           #Q_L2_max := #ZQ_L2_max / #MILLION / #THOUSAND;
           #Q_L3_max := #ZQ_L3_max / #MILLION / #THOUSAND;
   END_CASE;
   // calculate apparent energy unit     
   CASE #C_E_S_Unit OF
       1:
           IF ((#VEnergy_Meter_Unit[9] = TRUE) OR (#VEnergy_Meter_Unit[10] = TRUE)) THEN
               #S_Energy_Unit := 'kVAh';
               IF (#VEnergy_Meter_Unit[9] = FALSE) THEN
                   #E_Apparent_Rate1_Import := #ZE_Apparent_Rate1_Import / #THOUSAND;
               ELSE
                   #E_Apparent_Rate1_Import := #ZE_Apparent_Rate1_Import;
               END_IF;
               IF (#VEnergy_Meter_Unit[10] = FALSE) THEN
                   #E_Apparent_Rate2_Import := #ZE_Apparent_Rate2_Import / #THOUSAND;
               ELSE
                   #E_Apparent_Rate2_Import := #ZE_Apparent_Rate2_Import;
               END_IF;
           ELSE
               #S_Energy_Unit := 'VAh';
               #E_Apparent_Rate1_Import := #ZE_Apparent_Rate1_Import;
               #E_Apparent_Rate2_Import := #ZE_Apparent_Rate2_Import;
           END_IF;
       2:
           IF ((#VEnergy_Meter_Unit[9] = TRUE) OR (#VEnergy_Meter_Unit[10] = TRUE)) THEN
               #S_Energy_Unit := 'MVAh';
               IF (#VEnergy_Meter_Unit[9] = FALSE) THEN
                   #E_Apparent_Rate1_Import := #ZE_Apparent_Rate1_Import / #MILLION;
               ELSE
                   #E_Apparent_Rate1_Import := #ZE_Apparent_Rate1_Import / #THOUSAND;
               END_IF;
               IF (#VEnergy_Meter_Unit[10] = FALSE) THEN
                   #E_Apparent_Rate2_Import := #ZE_Apparent_Rate2_Import / #MILLION;
               ELSE
                   #E_Apparent_Rate2_Import := #ZE_Apparent_Rate2_Import / #THOUSAND;
               END_IF;
           ELSE
               #S_Energy_Unit := 'kVAh';
               #E_Apparent_Rate1_Import := #ZE_Apparent_Rate1_Import / #THOUSAND;
               #E_Apparent_Rate2_Import := #ZE_Apparent_Rate2_Import / #THOUSAND;
           END_IF;
       3:
           IF ((#VEnergy_Meter_Unit[9] = TRUE) OR (#VEnergy_Meter_Unit[10] = TRUE)) THEN
               #S_Energy_Unit := 'GVAh';
               IF (#VEnergy_Meter_Unit[9] = FALSE) THEN
                   #E_Apparent_Rate1_Import := #ZE_Apparent_Rate1_Import / #MILLION / #THOUSAND;
               ELSE
                   #E_Apparent_Rate1_Import := #ZE_Apparent_Rate1_Import / #MILLION;
               END_IF;
               IF (#VEnergy_Meter_Unit[10] = FALSE) THEN
                   #E_Apparent_Rate2_Import := #ZE_Apparent_Rate2_Import / #MILLION / #THOUSAND;
               ELSE
                   #E_Apparent_Rate2_Import := #ZE_Apparent_Rate2_Import / #MILLION;
               END_IF;
           ELSE
               #S_Energy_Unit := 'MVAh';
               #E_Apparent_Rate1_Import := #ZE_Apparent_Rate1_Import / #MILLION;
               #E_Apparent_Rate2_Import := #ZE_Apparent_Rate2_Import / #MILLION;
           END_IF;
       ELSE:
           IF ((#VEnergy_Meter_Unit[9] = TRUE) OR (#VEnergy_Meter_Unit[10] = TRUE)) THEN
               #S_Energy_Unit := 'TVAh';
               IF (#VEnergy_Meter_Unit[9] = FALSE) THEN
                   #E_Apparent_Rate1_Import := #ZE_Apparent_Rate1_Import / #MILLION / #MILLION;
               ELSE
                   #E_Apparent_Rate1_Import := #ZE_Apparent_Rate1_Import / #MILLION / #THOUSAND;
               END_IF;
               IF (#VEnergy_Meter_Unit[10] = FALSE) THEN
                   #E_Apparent_Rate2_Import := #ZE_Apparent_Rate2_Import / #MILLION / #MILLION;
               ELSE
                   #E_Apparent_Rate2_Import := #ZE_Apparent_Rate2_Import / #MILLION / #THOUSAND;
               END_IF;
           ELSE
               #S_Energy_Unit := 'GVAh';
               #E_Apparent_Rate1_Import := #ZE_Apparent_Rate1_Import / #MILLION / #THOUSAND;
               #E_Apparent_Rate2_Import := #ZE_Apparent_Rate2_Import / #MILLION / #THOUSAND;
           END_IF;
   END_CASE;
   // calculate active energy unit     
   CASE #C_E_P_Unit OF
       1:
           IF ((#VEnergy_Meter_Unit[1] = TRUE) OR (#VEnergy_Meter_Unit[2] = TRUE) OR
               (#VEnergy_Meter_Unit[3] = TRUE) OR (#VEnergy_Meter_Unit[4] = TRUE)) THEN
               #P_Energy_Unit := 'kWh';
               IF (#VEnergy_Meter_Unit[1] = FALSE) THEN
                   #E_Active_Rate1_Import := #ZE_Active_Rate1_Import / #THOUSAND;
               ELSE
                   #E_Active_Rate1_Import := #ZE_Active_Rate1_Import;
               END_IF;
               IF (#VEnergy_Meter_Unit[2] = FALSE) THEN
                   #E_Active_Rate2_Import := #ZE_Active_Rate2_Import / #THOUSAND;
               ELSE
                   #E_Active_Rate2_Import := #ZE_Active_Rate2_Import;
               END_IF;
               IF (#VEnergy_Meter_Unit[3] = FALSE) THEN
                   #E_Active_Rate1_Export := #ZE_Active_Rate1_Export / #THOUSAND;
               ELSE
                   #E_Active_Rate1_Export := #ZE_Active_Rate1_Export;
               END_IF;
               IF (#VEnergy_Meter_Unit[4] = FALSE) THEN
                   #E_Active_Rate1_Export := #ZE_Active_Rate1_Export / #THOUSAND;
               ELSE
                   #E_Active_Rate1_Export := #ZE_Active_Rate1_Export;
               END_IF;
           ELSE
               #P_Energy_Unit := 'Wh';
               #E_Active_Rate1_Import := #ZE_Active_Rate1_Import;
               #E_Active_Rate2_Import := #ZE_Active_Rate2_Import;
               #E_Active_Rate1_Export := #ZE_Active_Rate1_Export;
               #E_Active_Rate2_Export := #ZE_Active_Rate2_Export;
           END_IF;
       2:
           IF ((#VEnergy_Meter_Unit[1] = TRUE) OR (#VEnergy_Meter_Unit[2] = TRUE) OR
               (#VEnergy_Meter_Unit[3] = TRUE) OR (#VEnergy_Meter_Unit[4] = TRUE)) THEN
               #P_Energy_Unit := 'MWh';
               IF (#VEnergy_Meter_Unit[1] = FALSE) THEN
                   #E_Active_Rate1_Import := #ZE_Active_Rate1_Import / #MILLION;
               ELSE
                   #E_Active_Rate1_Import := #ZE_Active_Rate1_Import / #THOUSAND;
               END_IF;
               IF (#VEnergy_Meter_Unit[2] = FALSE) THEN
                   #E_Active_Rate2_Import := #ZE_Active_Rate2_Import / #MILLION;
               ELSE
                   #E_Active_Rate2_Import := #ZE_Active_Rate2_Import / #THOUSAND;
               END_IF;
               IF (#VEnergy_Meter_Unit[3] = FALSE) THEN
                   #E_Active_Rate1_Export := #ZE_Active_Rate1_Export / #MILLION;
               ELSE
                   #E_Active_Rate1_Export := #ZE_Active_Rate1_Export / #THOUSAND;
               END_IF;
               IF (#VEnergy_Meter_Unit[4] = FALSE) THEN
                   #E_Active_Rate2_Export := #ZE_Active_Rate2_Export / #MILLION;
               ELSE
                   #E_Active_Rate2_Export := #ZE_Active_Rate2_Export / #THOUSAND;
               END_IF;
           ELSE
               #P_Energy_Unit := 'kWh';
               #E_Active_Rate1_Import := #ZE_Active_Rate1_Import / #THOUSAND;
               #E_Active_Rate2_Import := #ZE_Active_Rate2_Import / #THOUSAND;
               #E_Active_Rate1_Export := #ZE_Active_Rate1_Export / #THOUSAND;
               #E_Active_Rate2_Export := #ZE_Active_Rate2_Export / #THOUSAND;
           END_IF;
       3:
           IF ((#VEnergy_Meter_Unit[1] = TRUE) OR (#VEnergy_Meter_Unit[2] = TRUE) OR
               (#VEnergy_Meter_Unit[3] = TRUE) OR (#VEnergy_Meter_Unit[4] = TRUE)) THEN
               #P_Energy_Unit := 'GWh';
               IF (#VEnergy_Meter_Unit[1] = FALSE) THEN
                   #E_Active_Rate1_Import := #ZE_Active_Rate1_Import / #MILLION / #THOUSAND;
               ELSE
                   #E_Active_Rate1_Import := #ZE_Active_Rate1_Import / #MILLION;
               END_IF;
               IF (#VEnergy_Meter_Unit[2] = FALSE) THEN
                   #E_Active_Rate2_Import := #ZE_Active_Rate2_Import / #MILLION / #THOUSAND;
               ELSE
                   #E_Active_Rate2_Import := #ZE_Active_Rate2_Import / #MILLION;
               END_IF;
               IF (#VEnergy_Meter_Unit[3] = FALSE) THEN
                   #E_Active_Rate1_Export := #ZE_Active_Rate1_Export / #MILLION / #THOUSAND;
               ELSE
                   #E_Active_Rate1_Export := #ZE_Active_Rate1_Export / #MILLION;
               END_IF;
               IF (#VEnergy_Meter_Unit[4] = FALSE) THEN
                   #E_Active_Rate2_Export := #ZE_Active_Rate2_Export / #MILLION / #THOUSAND;
               ELSE
                   #E_Active_Rate2_Export := #ZE_Active_Rate2_Export / #MILLION;
               END_IF;
           ELSE
               #P_Energy_Unit := 'MWh';
               #E_Active_Rate1_Import := #ZE_Active_Rate1_Import / #MILLION;
               #E_Active_Rate2_Import := #ZE_Active_Rate2_Import / #MILLION;
               #E_Active_Rate1_Export := #ZE_Active_Rate1_Export / #MILLION;
               #E_Active_Rate2_Export := #ZE_Active_Rate2_Export / #MILLION;
           END_IF;
       ELSE:
           IF ((#VEnergy_Meter_Unit[1] = TRUE) OR (#VEnergy_Meter_Unit[2] = TRUE) OR
               (#VEnergy_Meter_Unit[3] = TRUE) OR (#VEnergy_Meter_Unit[4] = TRUE)) THEN
               #P_Energy_Unit := 'TWh';
               IF (#VEnergy_Meter_Unit[1] = FALSE) THEN
                   #E_Active_Rate1_Import := #ZE_Active_Rate1_Import / #MILLION / #MILLION;
               ELSE
                   #E_Active_Rate1_Import := #ZE_Active_Rate1_Import / #MILLION / #THOUSAND;
               END_IF;
               IF (#VEnergy_Meter_Unit[2] = FALSE) THEN
                   #E_Active_Rate2_Import := #ZE_Active_Rate2_Import / #MILLION / #MILLION;
               ELSE
                   #E_Active_Rate2_Import := #ZE_Active_Rate2_Import / #MILLION / #THOUSAND;
               END_IF;
               IF (#VEnergy_Meter_Unit[3] = FALSE) THEN
                   #E_Active_Rate1_Export := #ZE_Active_Rate1_Export / #MILLION / #MILLION;
               ELSE
                   #E_Active_Rate1_Export := #ZE_Active_Rate1_Export / #MILLION / #THOUSAND;
               END_IF;
               IF (#VEnergy_Meter_Unit[4] = FALSE) THEN
                   #E_Active_Rate2_Export := #ZE_Active_Rate2_Export / #MILLION / #MILLION;
               ELSE
                   #E_Active_Rate2_Export := #ZE_Active_Rate2_Export / #MILLION / #THOUSAND;
               END_IF;
           ELSE
               #P_Energy_Unit := 'GWh';
               #E_Active_Rate1_Import := #ZE_Active_Rate1_Import / #MILLION / #THOUSAND;
               #E_Active_Rate2_Import := #ZE_Active_Rate2_Import / #MILLION / #THOUSAND;
               #E_Active_Rate1_Export := #ZE_Active_Rate1_Export / #MILLION / #THOUSAND;
               #E_Active_Rate2_Export := #ZE_Active_Rate2_Export / #MILLION / #THOUSAND;
           END_IF;
   END_CASE;
   // calculate reactive energy unit     
   CASE #C_E_Q_Unit OF
       1:
           IF ((#VEnergy_Meter_Unit[5] = TRUE) OR (#VEnergy_Meter_Unit[6] = TRUE) OR
               (#VEnergy_Meter_Unit[7] = TRUE) OR (#VEnergy_Meter_Unit[8] = TRUE)) THEN
               #Q_Energy_Unit := 'kWh';
               IF (#VEnergy_Meter_Unit[5] = FALSE) THEN
                   #E_Reactive_Rate1_Import := #ZE_Reactive_Rate1_Import / #THOUSAND;
               ELSE
                   #E_Reactive_Rate1_Import := #ZE_Reactive_Rate1_Import;
               END_IF;
               IF (#VEnergy_Meter_Unit[6] = FALSE) THEN
                   #E_Reactive_Rate2_Import := #ZE_Reactive_Rate2_Import / #THOUSAND;
               ELSE
                   #E_Reactive_Rate2_Import := #ZE_Reactive_Rate2_Import;
               END_IF;
               IF (#VEnergy_Meter_Unit[7] = FALSE) THEN
                   #E_Reactive_Rate1_Export := #ZE_Reactive_Rate1_Export / #THOUSAND;
               ELSE
                   #E_Reactive_Rate1_Export := #ZE_Reactive_Rate1_Export;
               END_IF;
               IF (#VEnergy_Meter_Unit[8] = FALSE) THEN
                   #E_Reactive_Rate2_Export := #ZE_Reactive_Rate2_Export / #THOUSAND;
               ELSE
                   #E_Reactive_Rate2_Export := #ZE_Reactive_Rate2_Export;
               END_IF;
           ELSE
               #Q_Energy_Unit := 'varh';
               #E_Reactive_Rate1_Import := #ZE_Reactive_Rate1_Import;
               #E_Reactive_Rate2_Import := #ZE_Reactive_Rate2_Import;
               #E_Reactive_Rate1_Export := #ZE_Reactive_Rate1_Export;
               #E_Reactive_Rate2_Export := #ZE_Reactive_Rate2_Export;
           END_IF;
       2:
           IF ((#VEnergy_Meter_Unit[5] = TRUE) OR (#VEnergy_Meter_Unit[6] = TRUE) OR
               (#VEnergy_Meter_Unit[7] = TRUE) OR (#VEnergy_Meter_Unit[8] = TRUE)) THEN
               #Q_Energy_Unit := 'MWh';
               IF (#VEnergy_Meter_Unit[5] = FALSE) THEN
                   #E_Reactive_Rate1_Import := #ZE_Reactive_Rate1_Import / #MILLION;
               ELSE
                   #E_Reactive_Rate1_Import := #ZE_Reactive_Rate1_Import;
               END_IF;
               IF (#VEnergy_Meter_Unit[6] = FALSE) THEN
                   #E_Reactive_Rate2_Import := #ZE_Reactive_Rate2_Import / #MILLION;
               ELSE
                   #E_Reactive_Rate2_Import := #ZE_Reactive_Rate2_Import;
               END_IF;
               IF (#VEnergy_Meter_Unit[7] = FALSE) THEN
                   #E_Reactive_Rate1_Export := #ZE_Reactive_Rate1_Export / #MILLION;
               ELSE
                   #E_Reactive_Rate1_Export := #ZE_Reactive_Rate1_Export;
               END_IF;
               IF (#VEnergy_Meter_Unit[8] = FALSE) THEN
                   #E_Reactive_Rate2_Export := #ZE_Reactive_Rate2_Export / #MILLION;
               ELSE
                   #E_Reactive_Rate2_Export := #ZE_Reactive_Rate2_Export;
               END_IF;
           ELSE
               #Q_Energy_Unit := 'kvarh';
               #E_Reactive_Rate1_Import := #ZE_Reactive_Rate1_Import / #THOUSAND;
               #E_Reactive_Rate2_Import := #ZE_Reactive_Rate2_Import / #THOUSAND;
               #E_Reactive_Rate1_Export := #ZE_Reactive_Rate1_Export / #THOUSAND;
               #E_Reactive_Rate2_Export := #ZE_Reactive_Rate2_Export / #THOUSAND;
           END_IF;
       3:
           IF ((#VEnergy_Meter_Unit[5] = TRUE) OR (#VEnergy_Meter_Unit[6] = TRUE) OR
               (#VEnergy_Meter_Unit[7] = TRUE) OR (#VEnergy_Meter_Unit[8] = TRUE)) THEN
               #Q_Energy_Unit := 'GWh';
               IF (#VEnergy_Meter_Unit[5] = FALSE) THEN
                   #E_Reactive_Rate1_Import := #ZE_Reactive_Rate1_Import / #MILLION / #THOUSAND;
               ELSE
                   #E_Reactive_Rate1_Import := #ZE_Reactive_Rate1_Import / #THOUSAND;
               END_IF;
               IF (#VEnergy_Meter_Unit[6] = FALSE) THEN
                   #E_Reactive_Rate2_Import := #ZE_Reactive_Rate2_Import / #MILLION / #THOUSAND;
               ELSE
                   #E_Reactive_Rate2_Import := #ZE_Reactive_Rate2_Import / #THOUSAND;
               END_IF;
               IF (#VEnergy_Meter_Unit[7] = FALSE) THEN
                   #E_Reactive_Rate1_Export := #ZE_Reactive_Rate1_Export / #MILLION / #THOUSAND;
               ELSE
                   #E_Reactive_Rate1_Export := #ZE_Reactive_Rate1_Export / #THOUSAND;
               END_IF;
               IF (#VEnergy_Meter_Unit[8] = FALSE) THEN
                   #E_Reactive_Rate2_Export := #ZE_Reactive_Rate2_Export / #MILLION / #THOUSAND;
               ELSE
                   #E_Reactive_Rate2_Export := #ZE_Reactive_Rate2_Export / #THOUSAND;
               END_IF;
           ELSE
               #Q_Energy_Unit := 'Mvarh';
               #E_Reactive_Rate1_Import := #ZE_Reactive_Rate1_Import / #MILLION;
               #E_Reactive_Rate2_Import := #ZE_Reactive_Rate2_Import / #MILLION;
               #E_Reactive_Rate1_Export := #ZE_Reactive_Rate1_Export / #MILLION;
               #E_Reactive_Rate2_Export := #ZE_Reactive_Rate2_Export / #MILLION;
           END_IF;
       ELSE:
           IF ((#VEnergy_Meter_Unit[5] = TRUE) OR (#VEnergy_Meter_Unit[6] = TRUE) OR
               (#VEnergy_Meter_Unit[7] = TRUE) OR (#VEnergy_Meter_Unit[8] = TRUE)) THEN
               #Q_Energy_Unit := 'TWh';
               IF (#VEnergy_Meter_Unit[5] = FALSE) THEN
                   #E_Reactive_Rate1_Import := #ZE_Reactive_Rate1_Import / #MILLION / #MILLION;
               ELSE
                   #E_Reactive_Rate1_Import := #ZE_Reactive_Rate1_Import / #MILLION / #THOUSAND;
               END_IF;
               IF (#VEnergy_Meter_Unit[6] = FALSE) THEN
                   #E_Reactive_Rate2_Import := #ZE_Reactive_Rate2_Import / #MILLION / #MILLION;
               ELSE
                   #E_Reactive_Rate2_Import := #ZE_Reactive_Rate2_Import / #MILLION / #THOUSAND;
               END_IF;
               IF (#VEnergy_Meter_Unit[7] = FALSE) THEN
                   #E_Reactive_Rate1_Export := #ZE_Reactive_Rate1_Export / #MILLION / #MILLION;
               ELSE
                   #E_Reactive_Rate1_Export := #ZE_Reactive_Rate1_Export / #MILLION / #THOUSAND;
               END_IF;
               IF (#VEnergy_Meter_Unit[8] = FALSE) THEN
                   #E_Reactive_Rate2_Export := #ZE_Reactive_Rate2_Export / #MILLION / #MILLION;
               ELSE
                   #E_Reactive_Rate2_Export := #ZE_Reactive_Rate2_Export / #MILLION / #THOUSAND;
               END_IF;
           ELSE
               #Q_Energy_Unit := 'Gvarh';
               #E_Reactive_Rate1_Import := #ZE_Reactive_Rate1_Import / #MILLION / #THOUSAND;
               #E_Reactive_Rate2_Import := #ZE_Reactive_Rate2_Import / #MILLION / #THOUSAND;
               #E_Reactive_Rate1_Export := #ZE_Reactive_Rate1_Export / #MILLION / #THOUSAND;
               #E_Reactive_Rate2_Export := #ZE_Reactive_Rate2_Export / #MILLION / #THOUSAND;
           END_IF;
   END_CASE;
   //======================================================================================================================
   //==========calculate scale final value=================================================================================
   //======================================================================================================================        
   // calculate scale final voltage PH-PH
   IF ((#AREA_TO_THOUSAND < #U_L1_L2_max) OR (#AREA_TO_THOUSAND < #U_L2_L3_max) OR (#AREA_TO_THOUSAND < #U_L3_L1_max)) THEN
       #ZScale_End_U_PH_PH := #ZSCALE_END_I4;
   ELSIF ((#AREA_TO_HUNDRED < #U_L1_L2_max) OR (#AREA_TO_HUNDRED < #U_L2_L3_max) OR (#AREA_TO_HUNDRED < #U_L3_L1_max)) THEN
       #ZScale_End_U_PH_PH := #ZSCALE_END_I3;
   ELSIF ((#AREA_TO_TEN < #U_L1_L2_max) OR (#AREA_TO_TEN < #U_L2_L3_max) OR (#AREA_TO_TEN < #U_L3_L1_max)) THEN
       #ZScale_End_U_PH_PH := #ZSCALE_END_I2;
   ELSIF ((0 <= #U_L1_L2_max) OR (0 <= #U_L2_L3_max) OR (0 <= #U_L3_L1_max)) THEN
       #ZScale_End_U_PH_PH := #ZSCALE_END_I1;
   ELSE
       ;
   END_IF;
   // selection maximum value
   #U_PH_PH := MAX(IN1 := #U_L1_L2_max, IN2 := #U_L2_L3_max, IN3 := #U_L3_L1_max, IN4 := 4.0);
   // 
   #Scale_End_U_PH_PH := (REAL_TO_DINT(#U_PH_PH * #FACTOR)) + (#ZScale_End_U_PH_PH - (REAL_TO_DINT(#U_PH_PH * #FACTOR) MOD #ZScale_End_U_PH_PH));
   // calculate scale final voltage PH-N
   IF ((#AREA_TO_THOUSAND < #U_L1_max) OR (#AREA_TO_THOUSAND < #U_L2_max) OR (#AREA_TO_THOUSAND < #U_L3_max)) THEN
       #ZScale_End_U_PH_N := #ZSCALE_END_I4;
   ELSIF ((#AREA_TO_HUNDRED < #U_L1_max) OR (#AREA_TO_HUNDRED < #U_L2_max) OR (#AREA_TO_HUNDRED < #U_L3_max)) THEN
       #ZScale_End_U_PH_N := #ZSCALE_END_I3;
   ELSIF ((#AREA_TO_TEN < #U_L1_max) OR (#AREA_TO_TEN < #U_L2_max) OR (#AREA_TO_TEN < #U_L3_max)) THEN
       #ZScale_End_U_PH_N := #ZSCALE_END_I2;
   ELSIF ((0 <= #U_L1_max) OR (0 <= #U_L2_max) OR (0 <= #U_L3_max)) THEN
       #ZScale_End_U_PH_N := #ZSCALE_END_I1;
   ELSE
       ;
   END_IF;
   // selection maximum value
   #U_PH_N := MAX(IN1 := #U_L1_max, IN2 := #U_L2_max, IN3 := #U_L3_max, IN4 := 4.0);
   // 
   #Scale_End_U_PH_N := (REAL_TO_DINT(#U_PH_N * #FACTOR)) + (#ZScale_End_U_PH_N - (REAL_TO_DINT(#U_PH_N * #FACTOR) MOD #ZScale_End_U_PH_N));
   // calculate scale final current
   IF ((#AREA_TO_THOUSAND < #I_L1_max) OR (#AREA_TO_THOUSAND < #I_L2_max) OR (#AREA_TO_THOUSAND < #I_L3_max)) THEN
       #ZScale_End_I := #ZSCALE_END_I4;
   ELSIF ((#AREA_TO_HUNDRED < #I_L1_max) OR (#AREA_TO_HUNDRED < #I_L2_max) OR (#AREA_TO_HUNDRED < #I_L3_max)) THEN
       #ZScale_End_I := #ZSCALE_END_I3;
   ELSIF ((#AREA_TO_TEN < #I_L1_max) OR (#AREA_TO_TEN < #I_L2_max) OR (#AREA_TO_TEN < #I_L3_max)) THEN
       #ZScale_End_I := #ZSCALE_END_I2;
   ELSIF ((0 <= #I_L1_max) OR (0 <= #I_L2_max) OR (0 <= #I_L3_max)) THEN
       #ZScale_End_I := #ZSCALE_END_I1;
   ELSE
       ;
   END_IF;
   // selection maximum value
   #I := MAX(IN1 := #I_L1_max, IN2 := #I_L2_max, IN3 := #I_L3_max, IN4 := 4.0);
   //
   #Scale_End_I := (REAL_TO_DINT(#I * #FACTOR)) + (#ZScale_End_I - (REAL_TO_DINT(#I * #FACTOR) MOD #ZScale_End_I));
   // calculate scale final apparent power    
   IF ((#AREA_TO_THOUSAND < #S_L1_max) OR (#AREA_TO_THOUSAND < #S_L2_max) OR
       (#AREA_TO_THOUSAND < #S_L3_max) OR (#AREA_TO_THOUSAND < #S_Total_max)) THEN
       #ZScale_End_S := #ZSCALE_END_SPQ4;
   ELSIF ((#AREA_TO_HUNDRED < #S_L1_max) OR (#AREA_TO_HUNDRED < #S_L2_max) OR
       (#AREA_TO_HUNDRED < #S_L3_max) OR (#AREA_TO_HUNDRED < #S_Total_max)) THEN
       #ZScale_End_S := #ZSCALE_END_SPQ3;
   ELSIF ((#AREA_TO_TEN < #S_L1_max) OR (#AREA_TO_TEN < #S_L2_max) OR
       (#AREA_TO_TEN < #S_L3_max) OR (#AREA_TO_TEN < #S_Total_max)) THEN
       #ZScale_End_S := #ZSCALE_END_SPQ2;
   ELSIF ((0 <= #S_L1_max) OR (0 <= #S_L2_max) OR (0 <= #S_L3_max) OR (0 <= #S_Total_max)) THEN
       #ZScale_End_S := #ZSCALE_END_SPQ1;
   ELSE
       ;
   END_IF;
   // selection maximum value 
   #S := MAX(IN1 := #S_L1_max, IN2 := #S_L2_max, IN3 := #S_L3_max, IN4 := #S_Total_max, IN5 := 4.0);
   //
   #Scale_End_S := (REAL_TO_DINT(#S * #FACTOR)) + (#ZScale_End_S - (REAL_TO_DINT(#S * #FACTOR) MOD #ZScale_End_S));
   // calculate scale final active power
   IF ((#AREA_TO_THOUSAND < #P_L1_max) OR (#AREA_TO_THOUSAND < #P_L2_max) OR
       (#AREA_TO_THOUSAND < #P_L3_max) OR (#AREA_TO_THOUSAND < #P_Total_max)) THEN
       #ZScale_End_P := #ZSCALE_END_SPQ4;
   ELSIF ((#AREA_TO_HUNDRED < #P_L1_max) OR (#AREA_TO_HUNDRED < #P_L2_max) OR
       (#AREA_TO_HUNDRED < #P_L3_max) OR (#AREA_TO_HUNDRED < #P_Total_max)) THEN
       #ZScale_End_P := #ZSCALE_END_SPQ3;
   ELSIF ((#AREA_TO_TEN < #P_L1_max) OR (#AREA_TO_TEN < #P_L2_max) OR
       (#AREA_TO_TEN < #P_L3_max) OR (#AREA_TO_TEN < #P_Total_max)) THEN
       #ZScale_End_P := #ZSCALE_END_SPQ2;
   ELSIF ((0 <= #P_L1_max) OR (0 <= #P_L2_max) OR (0 <= #P_L3_max) OR (0 <= #P_Total_max)) THEN
       #ZScale_End_P := #ZSCALE_END_SPQ1;
   ELSE
       ;
   END_IF;
   // selection maximum value
   #P := MAX(IN1 := #P_L1_max, IN2 := #P_L2_max, IN3 := #P_L3_max, IN4 := #P_Total_max, IN5 := 4.0);
   //
   #Scale_End_P := (REAL_TO_DINT(#P * #FACTOR)) + (#ZScale_End_P - (REAL_TO_DINT(#P * #FACTOR) MOD #ZScale_End_P));
   // calculate scale final reactive power max
   IF ((#AREA_TO_THOUSAND < #Q_L1_max) OR (#AREA_TO_THOUSAND < #Q_L2_max) OR
       (#AREA_TO_THOUSAND < #Q_L3_max) OR (#AREA_TO_THOUSAND < #Q_Total_max) OR
       (- #AREA_TO_THOUSAND > #Q_L1_min) OR (- #AREA_TO_THOUSAND > #Q_L2_min) OR
       (- #AREA_TO_THOUSAND > #Q_L3_min) OR (- #AREA_TO_THOUSAND > #Q_Total_min)) THEN
       #ZScale_End_Q := #ZSCALE_END_SPQ4;
   ELSIF ((#AREA_TO_HUNDRED < #Q_L1_max) OR (#AREA_TO_HUNDRED < #Q_L2_max) OR
       (#AREA_TO_HUNDRED < #Q_L3_max) OR (#AREA_TO_HUNDRED < #Q_Total_max) OR
       (- #AREA_TO_HUNDRED > #Q_L1_min) OR (- #AREA_TO_HUNDRED > #Q_L2_min) OR
       (- #AREA_TO_HUNDRED > #Q_L3_min) OR (- #AREA_TO_HUNDRED > #Q_Total_min)) THEN
       #ZScale_End_Q := #ZSCALE_END_SPQ3;
   ELSIF ((#AREA_TO_TEN < #Q_L1_max) OR (#AREA_TO_TEN < #Q_L2_max) OR
       (#AREA_TO_TEN < #Q_L3_max) OR (#AREA_TO_TEN < #Q_Total_max) OR
       (- #AREA_TO_TEN > #Q_L1_min) OR (- #AREA_TO_TEN > #Q_L2_min) OR
       (- #AREA_TO_TEN > #Q_L3_min) OR (- #AREA_TO_TEN > #Q_Total_min)) THEN
       #ZScale_End_Q := #ZSCALE_END_SPQ2;
   ELSIF ((0 <= #Q_L1_max) OR (0 <= #Q_L2_max) OR (0 <= #Q_L3_max) OR (0 <= #Q_Total_max) OR
       (0 >= #Q_L1_min) OR (0 >= #Q_L2_min) OR (0 >= #Q_L3_min) OR (0 >= #Q_Total_min)) THEN
       #ZScale_End_Q := #ZSCALE_END_SPQ1;
   ELSE
       ;
   END_IF;
   // calculate scale final reactive power max
   IF ((MAX(IN1 := #Q_L1_max, IN2 := #Q_L2_max, IN3 := #Q_L3_max, IN4 := #Q_Total_max)) = 0) THEN
       #Q := 4.0;
   ELSE
       #Q := MAX(IN1 := #Q_L1_max, IN2 := #Q_L2_max, IN3 := #Q_L3_max, IN4 := #Q_Total_max);
   END_IF;
   //
   IF (#Q > 0) THEN
       #Scale_End_Q := (REAL_TO_DINT(#Q * #FACTOR)) + (#ZScale_End_Q - (REAL_TO_DINT(#Q * #FACTOR) MOD #ZScale_End_Q));
   ELSIF (#Q < 0) THEN
       #Scale_End_Q := (REAL_TO_DINT(#Q * #FACTOR)) - (#ZScale_End_Q - (REAL_TO_DINT(#Q * #FACTOR) MOD #ZScale_End_Q));
   ELSE
       ;
   END_IF;
   // calculate scale final reactive power min
   IF ((MIN(IN1 := #Q_L1_min, IN2 := #Q_L2_min, IN3 := #Q_L3_min, IN4 := #Q_Total_min)) = 0) THEN
       #Q_min := -4.0;
   ELSE
       #Q_min := MIN(IN1 := #Q_L1_min, IN2 := #Q_L2_min, IN3 := #Q_L3_min, IN4 := #Q_Total_min);
   END_IF;
   //
   IF (#Q_min > 0) THEN
       #Scale_Begin_Q := 0;
   ELSIF (#Q_min < 0) THEN
       #Scale_Begin_Q := (REAL_TO_DINT(#Q_min * #FACTOR)) - (#ZScale_End_Q - (REAL_TO_DINT(#Q_min * #FACTOR) MOD #ZScale_End_Q));
   END_IF;
   //======================================================================================================================
   //==========value to output value=======================================================================================
   //======================================================================================================================
   // calculation value
   #Calculate_Value1 := #Driver_Data.Calculate_Value1;               // calculate value 1
   #Calculate_Value2 := #Driver_Data.Calculate_Value2;               // calculate value 2
   #Calculate_Value3 := #Driver_Data.Calculate_Value3;               // calculate value 3
   #Calculate_Value4 := #Driver_Data.Calculate_Value4;               // calculate value 4
   #Calculate_Value5 := #Driver_Data.Calculate_Value5;               // calculate value 5
   #Calculate_Value6 := #Driver_Data.Calculate_Value6;               // calculate value 6
   // selection of show modification
   #U_PH_PH_Mod := #Driver_Data.U_PH_PH_Mod;                    // voltage PH-PH show modification
   #U_PH_N_Mod := #Driver_Data.U_PH_N_Mod;                     // voltage PH-N show modification
   #I_Mod := #Driver_Data.I_Mod;                          // current show modification
   #S_Mod := #Driver_Data.S_Mod;                          // apparent power show modification
   #P_Mod := #Driver_Data.P_Mod;                          // active power show modification
   #Q_Mod := #Driver_Data.Q_Mod;                          // reactive power show modification
   #E_Mod := #Driver_Data.E_Mod;                          // energy meter show modification
   #f_Mod := #Driver_Data.f_Mod;                          // frequenz show modification
   #Cos_Mod := #Driver_Data.Cos_Mod;                        // efficiency factor show modification  
   // temp value to output value
   #f := #Zf;                                         // frequency
   #f_min := #Zf_min;                                     // minimum frequenz
   #f_max := #Zf_max;                                     // maximum frequenz
   #Cos_Total := #ZCos_Total;                                 // total efficiency factor
   #Cos_Total_min := #ZCos_Total_min;                             // minimum total efficiency factor
   #Cos_Total_max := #ZCos_Total_max;                             // maximum total efficiency factor
   #Cos_L1 := #ZCos_L1;                                    // efficiency factor L1       
   #Cos_L1_min := #ZCos_L1_min;                                // minimum efficiency factor L1
   #Cos_L1_max := #ZCos_L1_max;                                // maximum efficiency factor L1
   #Cos_L2 := #ZCos_L2;                                    // efficiency factor L2
   #Cos_L2_min := #ZCos_L2_min;                                // minimum efficiency factor L2
   #Cos_L2_max := #ZCos_L2_max;                                // maximum efficiency factor L2
   #Cos_L3 := #ZCOS_L3;                                    // efficiency factor L3
   #Cos_L3_min := #ZCos_L3_min;                                // minimum efficiency factor L3
   #Cos_L3_max := #ZCos_L3_max;                                // maximum efficiency factor L3
   // reset time Energy  
   #RTime_Data_Energy := #Driver_Data.RTime_Data_Energy;              // Reset Time
   #R_Year_Energy := BCD16_TO_INT(#ZRTime_Data_Energy[1]) + 100;      // Reset year   
   #R_Month_Energy := BCD16_TO_INT(#ZRTime_Data_Energy[2]) + 100;      // Reset month
   #R_Day_Energy := BCD16_TO_INT(#ZRTime_Data_Energy[3]) + 100;      // Reset day    
   #R_Hour_Energy := BCD16_TO_INT(#ZRTime_Data_Energy[4]) + 100;      // Reset hour   
   #R_Minute_Energy := BCD16_TO_INT(#ZRTime_Data_Energy[5]) + 100;      // Reset minute 
   #R_Second_Energy := BCD16_TO_INT(#ZRTime_Data_Energy[6]) + 100;      // Reset Second
   // reset time value
   #RTime_Data_Value := #Driver_Data.RTime_Data_Value;               // Reset Time
   #R_Year_Value := BCD16_TO_INT(#ZRTime_Data_Value[1]) + 100;       // Reset year   
   #R_Month_Value := BCD16_TO_INT(#ZRTime_Data_Value[2]) + 100;       // Reset month  
   #R_Day_Value := BCD16_TO_INT(#ZRTime_Data_Value[3]) + 100;       // Reset day    
   #R_Hour_Value := BCD16_TO_INT(#ZRTime_Data_Value[4]) + 100;       // Reset hour   
   #R_Minute_Value := BCD16_TO_INT(#ZRTime_Data_Value[5]) + 100;       // Reset minute 
   #R_Second_Value := BCD16_TO_INT(#ZRTime_Data_Value[6]) + 100;       // Reset Second
   // HMI_Bits
   IF (#Driver_Data.Rest_Start_Auto = TRUE) THEN
       #Start_Auto := FALSE;
       #Start_Acyclic := FALSE;
   ELSE
       ;
   END_IF;
   #HMI_Bits.Start_Acyclic := #Start_Acyclic;
   #HMI_Bits.Start_Auto := #Start_Auto;
   #HMI_Bits.Reset_min_max_Data := #Reset_min_max_Data;
   #HMI_Bits.Reset_Energy_Meter := #Reset_Energy_Meter;
   //
   #Read_Value := #Driver_Data.Read_Value;
   //======================================================================================================================
   //==========error code==================================================================================================
   //======================================================================================================================  
   // error code output
   #ERROR := #Fehler;
END_FUNCTION_BLOCK
